FUNCTION_BLOCK INTERNAL FINAL FB_WriteRepeatedFieldUint32Tests EXTENDS FB_TestSuite
VAR_INPUT
END_VAR
VAR_OUTPUT
END_VAR
VAR
	fbFieldCodec : FB_FieldCodecUInt32(nTag:= 0);
	aActual    	 : ARRAY [0..7] OF UDINT;
	fbRepeatedField		: FB_RepeatedField(anyArray:= F_ToAnyType(aActual), anyFirstElem:= F_ToAnyType(aActual[0]), ipFieldCodec:= fbFieldCodec);
END_VAR

ShouldWriteRepeatedFieldTheory();

METHOD PRIVATE Reset
VAR_INPUT
END_VAR
fbRepeatedField.Initialize();
MEMSET(destAddr:= ADR(aActual), fillByte:= 16#0, n:= SIZEOF(aActual));
END_METHOD

METHOD PRIVATE ShouldWriteRepeatedField
VAR_IN_OUT CONSTANT
    aExpected   : ARRAY [*] OF BYTE;
END_VAR
VAR_INPUT
    aValues     : ARRAY [0..7] OF UDINT;
    nLength     : UDINT;
    nTag        : UDINT;
    nBufferPosStart     : UDINT;
    nExpectedBufferPos  : UDINT;
    ipFieldCodec        : I_FieldCodec;
END_VAR
VAR_INST
    fbCtx   : FB_WriteContext;
END_VAR
VAR
    aActualBuffer       : ARRAY [0..63] OF BYTE;
    hr                  : HRESULT;

END_VAR
// Arrange
Reset();
fbCtx.FromBuffer(aActualBuffer);
fbCtx.refCtx.stState.nBufferPos := nBufferPosStart;
ipFieldCodec.Tag := nTag;
fbRepeatedField.InitializeFromArray(anyArray:= F_ToAnyType(aValues), anyFirstElem:= F_ToAnyType(aValues[0]), nCount:= nLength);

// Act
hr := fbRepeatedField.WriteTo(fbWriteCtx:= fbCtx, ipFieldCodec:= ipFieldCodec);

// Assert
AssertEquals_DINT(
    Expected:= S_OK,
    Actual:= hr,
    Message:= 'Expected S_OK instead of error');
    
{warning disable C0041}
AssertArrayEquals_BYTE(Expecteds:= aExpected, Actuals:= aActualBuffer, Message:= '');
 
AssertEquals_UDINT(
    Expected:= nExpectedBufferPos,
    Actual:= fbCtx.refCtx.stState.nBufferPos,
    Message:= CONCAT('Expected stState.nBufferPos to equal ', TO_STRING(nExpectedBufferPos)));
END_METHOD

METHOD PRIVATE ShouldWriteRepeatedFieldTheory : REFERENCE TO FB_Test
VAR CONSTANT
    cRawValueZeroLength     : ARRAY[0..63] OF BYTE := [16#00, 16#00];
    cRawValue1              : ARRAY[0..63] OF BYTE := [16#00, 16#0A, 16#07, 16#00, 16#01, 16#FF, 16#01, 16#96, 16#01, 16#04];  
END_VAR

VAR CONSTANT
    aExpectedZeroLength     : ARRAY [0..7] OF UDINT := [0, 0, 0, 0, 0, 0, 0, 0];
    aExpected1              : ARRAY [0..7] OF UDINT := [0, 1, 255, 150, 4, 0, 0, 0];
END_VAR
TEST(__POUNAME());

ShouldWriteRepeatedField(aExpected:= cRawValueZeroLength, aValues:= aExpectedZeroLength, nLength:= 0, nTag:= F_MakeTag(1, E_WireType.LengthDelimited), nBufferPosStart:= 0, nExpectedBufferPos:= 0, ipFieldCodec:= THIS^.fbFieldCodec);
ShouldWriteRepeatedField(aExpected:= cRawValue1, aValues:= aExpected1, nLength:= 5, nTag:= F_MakeTag(1, E_WireType.LengthDelimited), nBufferPosStart:= 1, nExpectedBufferPos:= 10, ipFieldCodec:= THIS^.fbFieldCodec);

TEST_FINISHED_NAMED(__POUNAME());
END_METHOD

END_FUNCTION_BLOCK

(* stored: Version 1.1.0.1
   POU FB_WriteRepeatedFieldUint32Tests: Id {91b1b011-0625-4ddf-9329-2c0e21f587c3}, SpecialFunc None
   Method Reset: Id {4a025e58-9fe7-49ad-a4be-8d606c3f4970}
   Method ShouldWriteRepeatedField: Id {4208354a-28e1-4c49-a33a-7498f97fbfa9}
   Method ShouldWriteRepeatedFieldTheory: Id {0ec15e55-0326-40c9-b1d0-5419d52a963e} *)
